Universal Robots PolyScope program: ad_lab_exe_2_2_34.urp

Program ad_lab_exe_2_2_34 (createdIn=3.2.19293 lastSavedIn=3.2.19293 directory=/programs installation=default robotSerialNumber=2015351391)
Calibrated DH parameters: a=[0.000352, -0.161198, -0.373486, 0.00005, 0.000049, 0]; d=[0.089268, 352.477598, -320.08558, -32.281492, 0.094939, 0.082518]; alpha=[1.570728, 0.001116, -0.003686, 1.571189, -1.570572, 0]; deltaTheta=[-0.000012, 1.181849, -1.491165, 0.309495, -0.000007, 0.000025]
Robot Program (runOnlyOnce=false motionType=MoveJ speed=1.047198 acceleration=1.396263 recalculateMotions=false)
  current_pos := get_actual_tcp_pose()
  length_1 :=  (valueSource=Operator message=please input length: valueType=Float)
  offset_b := p[length_1,0,0,0,0,0]
  offset_c := p[length_1,0,-length_1,0,0,0]
  offset_d := p[0,0,-length_1,0,0,0]
  pos_b := pose_trans(current_pos,offset_b)
  pos_c := pose_trans(current_pos,offset_c)
  pos_d := pose_trans(current_pos,offset_d)
  MoveL speed 250 mm/s, acceleration 1200 mm/s^2 (recalculateMotions=false) feature=Base
    Waypoint 路点 (Variable): variable=current_pos
    Waypoint 路点 (Variable): variable=pos_b
    Waypoint 路点 (Variable): variable=pos_c
    Waypoint 路点 (Variable): variable=pos_d
    Waypoint 路点 (Variable): variable=current_pos
